FUNCTION_BLOCK FB_PortRack EXTENDS FB_Rack

VAR
END_VAR

METHOD FB_init : BOOL
VAR_INPUT
	bInitRetains : BOOL; // if TRUE, the retain variables are initialized (warm start / cold start)
	bInCopyCode : BOOL;  // if TRUE, the instance afterwards gets moved into the copy code (online change)
END_VAR
eObjectType := E_ObjectType.OBJECTTYPE_PortRack;
eObjectGroup := E_ObjectGroup.OBJECTGROUP_Target OR E_ObjectGroup.OBJECTGROUP_Rack;
END_METHOD

METHOD M_AddChild : ERRORID
VAR_INPUT
	pObject : POINTER TO FB_Object;
	nSlotNr	: UINT;
	nIndex 	: INT;
END_VAR
//Kann folgende Objekte aufnehmen:
//Point, Ports
IF pObject > 0 THEN
	IF pObject^.P_eObjectType = E_ObjectType.OBJECTTYPE_Point THEN
		M_AddChild := SUPER^.M_AddChild(pObject,nSlotNr,nIndex);
	ELSIF pObject^.P_eObjectType = E_ObjectType.OBJECTTYPE_Port THEN
		//darf nur in ein Slot
		IF nSlotNr > 0 THEN
			M_AddChild := SUPER^.M_AddChild(pObject,nSlotNr,nIndex);
		ELSE
			M_AddChild := E_ErrorIdObjMgmt.ERRORID_InvalidSlotNumber;	
		END_IF
	ELSE
		M_AddChild := E_ErrorIdObjMgmt.ERRORID_InvalidParentObject;
	END_IF
ELSE
	M_AddChild := E_ErrorIdObjMgmt.ERRORID_InvalidParentObject;
END_IF
END_METHOD

METHOD M_CheckAction : ERRORID
VAR_INPUT
	refActionData 	: REFERENCE TO ST_ActionData;
	pCorrelObject	: POINTER TO FB_Object;
END_VAR

VAR
END_VAR
END_METHOD

END_FUNCTION_BLOCK

(* stored: Version 1.1.0.1, ProductVersion 3.1.4022.18
   POU FB_PortRack: Id {62d6526b-96b8-4d33-9998-28b6093b3058}, SpecialFunc None
   Method FB_init: Id {7f470861-152b-4752-bff1-37c03565f42e}
   Method M_AddChild: Id {4de6bc23-1f09-448c-871e-62a4c25a4837}
   Method M_CheckAction: Id {e7c90908-6c0f-4d13-89c0-49048327fa37} *)
